FUNCTION POU : BOOL
VAR_INPUT
  Huidige_tijd : INT; //Invoer van de tijd
END_VAR

IF (Huidige_tijd >= 0) AND (Huidige_tijd <= 2400) THEN
	IF Huidige_tijd >= 1000 THEN
		POU := TRUE; // Order is klaar voor transport
	ELSE
		POU := FALSE; // Order is niet klaar voor transport
	END_IF
ELSE
	POU := FALSE; //Geeft aan dat de ingevoerde tijd ongeldig is
END_IF

END_FUNCTION

(* stored: Version 1.1.0.1, ProductVersion 3.1.4024.12
   POU POU: Id {7365f783-f984-4baf-ae0c-23fcb59f0d1e}, SpecialFunc None *)
